Yaskawa INFORM job: SAMPLE.JBI

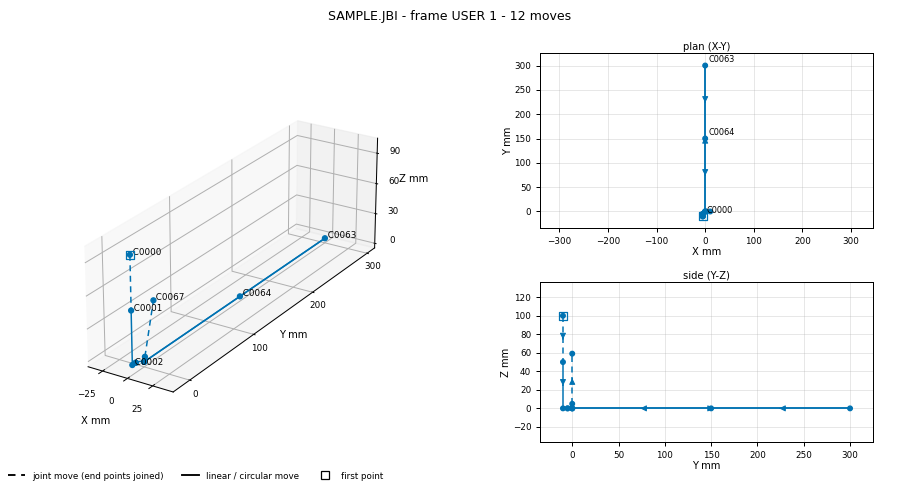
[picture p0: tool path of SAMPLE.JBI in frame USER 1, 12 of 13 moves have a stored position in this frame; points joined in program order, loops and branches not executed]
/JOB
//NAME BTEST
//POS
///NPOS 68,0,0,0,0,0
///USER 1
///TOOL 8
///POSTYPE USER
///RECTAN
///RCONF 0,0,0,0,0,0,0,0
C0000=-5.000,-10.000,100.000,180.000,0.000,-45.000
C0001=-5.000,-10.000,50.000,180.000,0.000,-45.000
C0002=-5.000,-10.000,0.000,180.000,0.000,-45.000
C0003=-5.000,-5.000,0.000,180.000,0.000,-45.000
C0004=-5.000,-5.000,0.000,180.000,0.000,-45.000
C0005=-3.536,-1.464,0.000,180.000,0.000,-45.000
C0006=0.000,0.000,0.000,180.000,0.000,-45.000
C0007=0.000,0.000,0.000,180.000,0.000,-45.000

(...)
///TOOL 9
(...)
C0062=150.000,300.000,0.000,-172.893,7.053,-44.561
C0063=0.000,300.000,0.000,172.893,7.053,-45.439
C0064=0.000,150.000,0.000,172.893,7.053,-45.439
C0065=0.000,0.000,0.000,172.893,7.053,-45.439
C0066=0.868,0.000,4.924,172.893,7.053,-45.439
C0067=10.419,0.000,59.088,172.893,7.053,-45.439
//INST
///DATE 2016/12/13 15:45
///COMM BY-ROBOTMASTER
///ATTR SC,RW,RJ
////FRAME USER 1
///GROUP1 RB1
NOP
CALL JOB:TOOL1
CALL JOB:APPROACH
MOVJ C0000 VJ=50.0
MOVJ C0001 VJ=50.0
MOVL C0002 V=50.0
CALL JOB:TOOLON
MOVL C0003 V=50.0
MOVC C0004 V=50.0
MOVC C0005 V=50.0
MOVC C0006 V=50.0
MOVL C0007 V=50.0

(...)

MOVL C0063 V=50.0
MOVL C0064 V=50.0
MOVL C0065 V=50.0
CALL JOB:TOOLOFF
MOVJ C0066 VJ=50.0
MOVJ C0067 VJ=50.0
CALL JOB:RETRACT
END
